{attribute 'qualified_only'}
{attribute 'strict'}
TYPE AxisStatus :
(
	Ready,
	STO_Active,
	Faulted
);
END_TYPE

(* stored: Version 1.1.0.1, ProductVersion 3.1.4024.13
   DUT AxisStatus: Id {b6b19266-60ab-4664-95b4-febab0c3e648} *)
